// TIA Portal V20 export
DATA_BLOCK "temp_db_for_test"   // DB372
// stored: MemoryReserve 100, Namespace Unit1.Em5
   VAR
      statJR_PnP_RnR : Struct
         currentCount : Int;
         processCount : Int;
         Ongoing : Bool;
         Complete : Bool;
      END_STRUCT;
   END_VAR
BEGIN
END_DATA_BLOCK
